{attribute addProperty BoxType "ELX3351-0000-0016"}
{attribute addProperty Id "StatusAT %I*Status_CB0A06B3162"}
{attribute addProperty CRC "3101727874"}
{attribute addProperty SizeInBites "16"}
{attribute addProperty SizeInBytes "2"}
TYPE RMB_Status_B8E09C82 :
STRUCT
	{attribute addProperty Name "Status"}
	Status AT %I* : Status_CB0A06B3;
END_STRUCT
END_TYPE

(* stored: Version 1.2.0.0, ProductVersion 3.1.4024.9
   DUT RMB_Status_B8E09C82: Id {a5d3e48a-8858-402d-b55a-7e0553c9b8ee} *)
